Staubli VAL3: printScroll.pgx

program printScroll(screen& x_scr)
  local num i
  local num lX
  local num lY
begin
  //-----------------------------------------------------------------------
  //Header begin
  //Description of program
  //  Put the scrool on the right of the list menu.
  // 在列表菜单右边放滚动条
  //History
  //  Creation : 28-04-08 - f.Rob
  //
  //Example
  //  call printScroll(scrMy)
  //
  //  Modified : 08-08-22 - J.Cook     Add screen parameter
  //Header end
  //-----------------------------------------------------------------------
  if size(sItems)>nBottomY
    //Find the percentage
    //Windows style
    //i=(size(sItems)-nBottomY+1)/(nFirst+1)
    // nokia style
    i=(size(sItems))/(nFirst+nView+1)
    lX=nTopX+nBottomX+1
    lY=roundUp((nBottomY)/i+nTopY)
    for i=nTopY+1 to nBottomY
      gotoxy(x_scr, lX,i)
      if i==lY
        //
        put(x_scr, "■")
        //
      else
        put(x_scr, "│")
      endIf
    endFor
  endIf
end
